// TwinCAT 3 PLC project Untitled2
// ProgramVersion: 3.1.4024.0
// libraries:
//   Tc2_Standard, * (Beckhoff Automation GmbH)
//   Tc2_System, * (Beckhoff Automation GmbH)
//   Tc3_Module, * (Beckhoff Automation GmbH)
//   VisuSymbols,3.5.10.0,System
// project tree:
//   / CoffeeMakerTask.TcTTO, GlobalTextList.TcGTLO, PlcTask.TcTTO, ResetTask.TcTTO, TaksLightsON.TcTTO, Visualization Manager.TcVMO (not stored)
//   POUs/ CoffeeMaker.TcPOU, DayOfWeek.TcPOU, GVL.TcGVL, IsItAWorkDay.TcPOU, LightsON.TcPOU, MAIN.TcPOU, Reset.TcPOU, Visualization.TcVIS
// real-time tasks:
//   TASK PlcTask: cycle T#10ms, priority 1, ADS port 350
//   TASK CoffeeMakerTask: cycle T#10ms, priority 2, ADS port 351
//   TASK TaksLightsON: cycle T#10ms, priority 3, ADS port 352
//   TASK ResetTask: cycle T#10ms, priority 4, ADS port 353

CONFIGURATION Untitled2
    RESOURCE PLC ON TwinCAT3
        TASK CoffeeMakerTask(INTERVAL := T#10ms, PRIORITY := 2);
        TASK PlcTask(INTERVAL := T#10ms, PRIORITY := 1);
        TASK ResetTask(INTERVAL := T#10ms, PRIORITY := 4);
        TASK TaksLightsON(INTERVAL := T#10ms, PRIORITY := 3);
        PROGRAM CoffeeMaker WITH CoffeeMakerTask : CoffeeMaker;
        PROGRAM MAIN WITH PlcTask : MAIN;
        PROGRAM Reset WITH ResetTask : Reset;
        PROGRAM LightsON WITH TaksLightsON : LightsON;
    END_RESOURCE
END_CONFIGURATION

// ---- POUs/GVL.TcGVL
{attribute 'qualified_only'}
VAR_GLOBAL
	bSetAlarm : BOOL := FALSE;			//Triggers the alarm to start the routine
	bAlarmON : BOOL := FALSE;			//Indicates if the alarm is currently active
	bWorkDayStatus : BOOL := FALSE;		//Indicates if the current day is a workday
	bCoffeeReady : BOOL := FALSE;		//Indicates if the coffee is ready
	bLightsON : BOOL := FALSE;			//Indicates if the lights are on
	bReset: BOOL;						//Triggers a reset of the system
	bBrewing: BOOL := FALSE;			//Indicates if coffee is brewing
	
	LightDelayTimer : TON;				//Timer for delaying light activation after the alarm goes off
	ResetTimer: TON;					//Timer to introduce a delay during reset.
	AlarmTimer : TON;					//Timer controlling when the alarm goes off.
	CoffeeTimer : TON;
	tCoffeeTime : TIME := T#15S;		//Duration before coffee is ready
	tLightDelayTime : TIME := T#3S;		//Delay time before lights turn of after the alarm goes off
	AlarmTime : TIME :=T#1S; 			//Time till alarm goes off
	
	DayCounter : INT := 0; 				//Counts the day (1-7)
	
	TheDayOfWeek : STRING[10] := '' ;	//Holds the current day of the week as text
	
END_VAR

// ---- POUs/CoffeeMaker.TcPOU
PROGRAM CoffeeMaker

VAR

END_VAR

//Checks if both the alarm and the lights are on and if its a workday, coffee will be made
IF (GVL.bAlarmON AND GVL.bLightsON AND GVL.bWorkDayStatus) THEN
	GVL.CoffeeTimer(IN := TRUE, PT := GVL.tCoffeeTime); //Starting the timer with the predefined time
ELSE
	GVL.CoffeeTimer(IN := FALSE);
	GVL.bCoffeeReady := FALSE;
END_IF

//Indicates if coffee is brewing
IF GVL.CoffeeTimer.IN THEN
	GVL.bBrewing := TRUE;
	ELSE
	GVL.bBrewing := FALSE;
END_IF

//Indicates that the coffee is ready when the timer is finished
IF GVL.CoffeeTimer.Q THEN
	GVL.bCoffeeReady := TRUE;
	GVL.bBrewing := FALSE;
END_IF

END_PROGRAM

// ---- POUs/MAIN.TcPOU
PROGRAM MAIN

VAR
	
END_VAR

//Milan Oude Nijeweme
//517922
//Process and Safety individual assignment

//This program provides a structured morning routine where, in sequence, an alarm goes off,
//lights turn on, and coffee is made. it accounts for the day of the week to determine if
//it's a workday and includes a reset feature to restore all actions and prepare for the
//next routine.


//Ceck if the alarm is set and is currently off
IF GVL.bSetAlarm AND NOT GVL.bAlarmON THEN
		GVL.AlarmTimer(IN := TRUE, PT := GVL.AlarmTime); //Starts the timer for the alarm with the predefined time
			IF GVL.AlarmTimer.Q THEN
				GVL.bAlarmON := TRUE;
		 
				GVL.DayCounter := GVL.DayCounter + 1; //Keeps track of day changes
		
					IF GVL.DayCounter > 7 THEN //Reset DayCounter to 1 if it exceeds 7 so its a weekly cycle
						GVL.DayCounter := 1;
					END_IF
			
				GVL.AlarmTimer(IN := FALSE);
				gvl.bSetAlarm := FALSE;	
			END_IF
END_IF

//Determine if it's a workday based on the current day
GVL.bWorkDayStatus := IsItAWorkDay(GVL.DayCounter);

//Gives the name of the day 
GVL.TheDayOfWeek := DayOfWeek(GVL.DayCounter);

END_PROGRAM

// ---- POUs/IsItAWorkDay.TcPOU
FUNCTION IsItAWorkDay : BOOL

VAR_INPUT
	Day : INT; //Current Day
END_VAR



//Checks if the day of the week is a workday
IF GVL.DayCounter >= 1 AND GVL.DayCounter <= 5 THEN
    IsItAWorkDay := TRUE; //Workday (Monday till friday)
ELSE
    IsItAWorkDay := FALSE; // Weekend (Saturday and sunday)
END_IF

END_FUNCTION

// ---- POUs/DayOfWeek.TcPOU
FUNCTION DayOfWeek : STRING

VAR_INPUT
	Day : INT; //Current day of the week
END_VAR

//transfers int to text for the visualization
CASE Day OF
	1: DayOfWeek := 'Maandag';
	2: DayOfWeek := 'Dinsdag';
	3: DayOfWeek := 'Woensdag';
	4: DayOfWeek := 'Donderdag';
	5: DayOfWeek := 'Vrijdag';
	6: DayOfWeek := 'Zaterdag';
	7: DayOfWeek := 'Zondag';
END_CASE

END_FUNCTION

// ---- POUs/Reset.TcPOU
PROGRAM Reset
VAR
END_VAR

//Resets all the variables so the alarm can be set again.
IF GVL.bReset THEN
	GVL.ResetTimer(IN:=TRUE, PT := T#1S);
	IF GVL.ResetTimer.Q THEN
		GVL.LightDelayTimer(IN:=FALSE);
		GVL.bAlarmON := FALSE;
		GVL.bLightsON := FALSE;
		GVL.bCoffeeReady := FALSE;
		GVL.bReset := FALSE;
		GVL.ResetTimer(IN:=FALSE);
	END_IF
END_IF

END_PROGRAM

// ---- POUs/LightsON.TcPOU
PROGRAM LightsON

VAR
	
END_VAR

//Truns lights on when alarm goes off
IF GVL.bAlarmON THEN
	GVL.LightDelayTimer(IN:=TRUE, PT := GVL.tLightDelayTime); //Makes sure the alarm goes off after a predefined delay
		IF GVL.LightDelayTimer.Q THEN
			GVL.bLightsON := TRUE;
		END_IF
ELSE
	GVL.bLightsON := FALSE;
END_IF

END_PROGRAM

// ---- GlobalTextList.TcGTLO
TEXTLIST GlobalTextList
  570 = '%i'
  439 = '%s'
  717 = 'AlarmON'
  901 = 'Coffee Brewing'
  724 = 'CoffeeReady'
  97 = 'Day of the week'
  994 = 'Desired'
  143 = 'Desired temperature'
  324 = 'Door closed'
  176 = 'LightsON'
  816 = 'Reset'
  892 = 'sdfsf '
  481 = 'Set Alarm'
  913 = 'Set alarm over 10 seconds'
  654 = 'Shower'
  677 = 'Start Routine'
  52 = 'Tap open'
END_TEXTLIST

// ---- POUs/Visualization.TcVIS
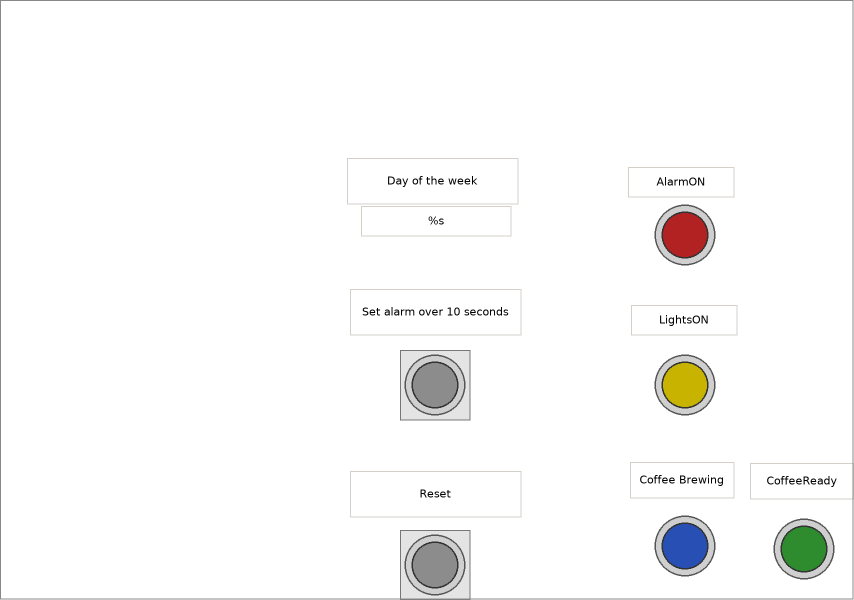
VISUALIZATION Visualization  // 854x600
    Lamp1 (650,200 70x70), variable: GVL.bAlarmON, style: Lamp-Lamp1-Red
    Lamp1 (650,350 70x70), variable: GVL.bLightsON, style: Lamp-Lamp1-Yellow
    Lamp1 (650,511 70x70), variable: GVL.bBrewing, style: Lamp-Lamp1-Blue
    Textfield (628,167 106x30), "AlarmON"
    Textfield (631,305 106x30), "LightsON"
    Textfield (630,462 104x36), "Coffee Brewing"
    Textfield (361,206 150x30), "%s", text variable: GVL.TheDayOfWeek
    PushSwitch (400,350 70x70), variable: GVL.bSetAlarm, behaviour: TOGGLE, style: Switch-PushSwitch-Gray
    Textfield (350,289 171x46), "Set alarm over 10 seconds"
    PushSwitch (400,530 70x70), variable: GVL.bReset, behaviour: TOGGLE, style: Switch-PushSwitch-Gray
    Textfield (350,471 171x46), "Reset"
    Textfield (347,158 171x46), "Day of the week"
    Textfield (750,463 104x36), "CoffeeReady"
    Lamp1 (769,514 70x70), variable: GVL.bCoffeeReady, style: Lamp-Lamp1-Green
END_VISUALIZATION
